ABB RobotStudio station: Example_station.rsstn

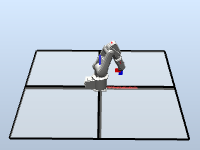
Station First (saved by RobotStudio 6.7.7936.1011)
Controller MTRN4230
  mechanical unit ROB_1: IRB120_3_58__01, 6 joints, base frame (0, 0, 0) mm
Layout (positions relative to the parent item):
  - IRB120_3_58__01 [mechanism, from Robots\IRB120_3_58_G_01.rslib] at (0, 0, 0) mm; joint values [0.3488, 0.4268, 0.7489, 0, 0.3951, 0.3488] (rad or m)
